// TIA Portal V18 export
FUNCTION_BLOCK "Source_select"   // FB1, FBD
TITLE = Source selection
{ S7_Optimized_Access := 'TRUE' }
VERSION : 0.1
// Source select
// stored: AutoNumber true, IsIECCheckEnabled false, IsRetainMemResEnabled false, MemoryReserve 100, SetENOAutomatically false, UDAEnableTagReadback false
   VAR_INPUT
      START : Bool;
      SP : Real;
      PV : Real;
      COUNTER_SP : Real;
      CHW_CT_SP : Real;
      CT_HW_SP : Real;
      HW_STEAM_SP : Real;
      CT_CHW_SP : Real;
      CHW_CHBr_SP : Real;
   END_VAR
   VAR_OUTPUT
      SOURCE_SEL : Int;
      STATUS : Word;
   END_VAR
   VAR
      Heating : Int;
      Cooling : Int;
      SUB_SP_COUNTER_SP : Real;
      ADD_SP_COUNTER_SP : Real;
      SS_TP1 { S7_SetPoint := 'True'} : TP_TIME;
      SS_TP2 { S7_SetPoint := 'True'} : TP_TIME;
      SS_TP3 { S7_SetPoint := 'True'} : TP_TIME;
      SS_TP4 { S7_SetPoint := 'True'} : TP_TIME;
      SS_TP5 { S7_SetPoint := 'True'} : TP_TIME;
      SS_TP6 { S7_SetPoint := 'True'} : TP_TIME;
      SS_TON1 { S7_SetPoint := 'True'} : TON_TIME;
      SS_TON3 { S7_SetPoint := 'True'} : TON_TIME;
      SS_TON4 { S7_SetPoint := 'True'} : TON_TIME;
      SS_TON5 { S7_SetPoint := 'True'} : TON_TIME;
      SS_TON6 { S7_SetPoint := 'True'} : TON_TIME;
      SS_TON7 { S7_SetPoint := 'True'} : TON_TIME;
   END_VAR
BEGIN

REGION Network 1: Heating
   // Heating
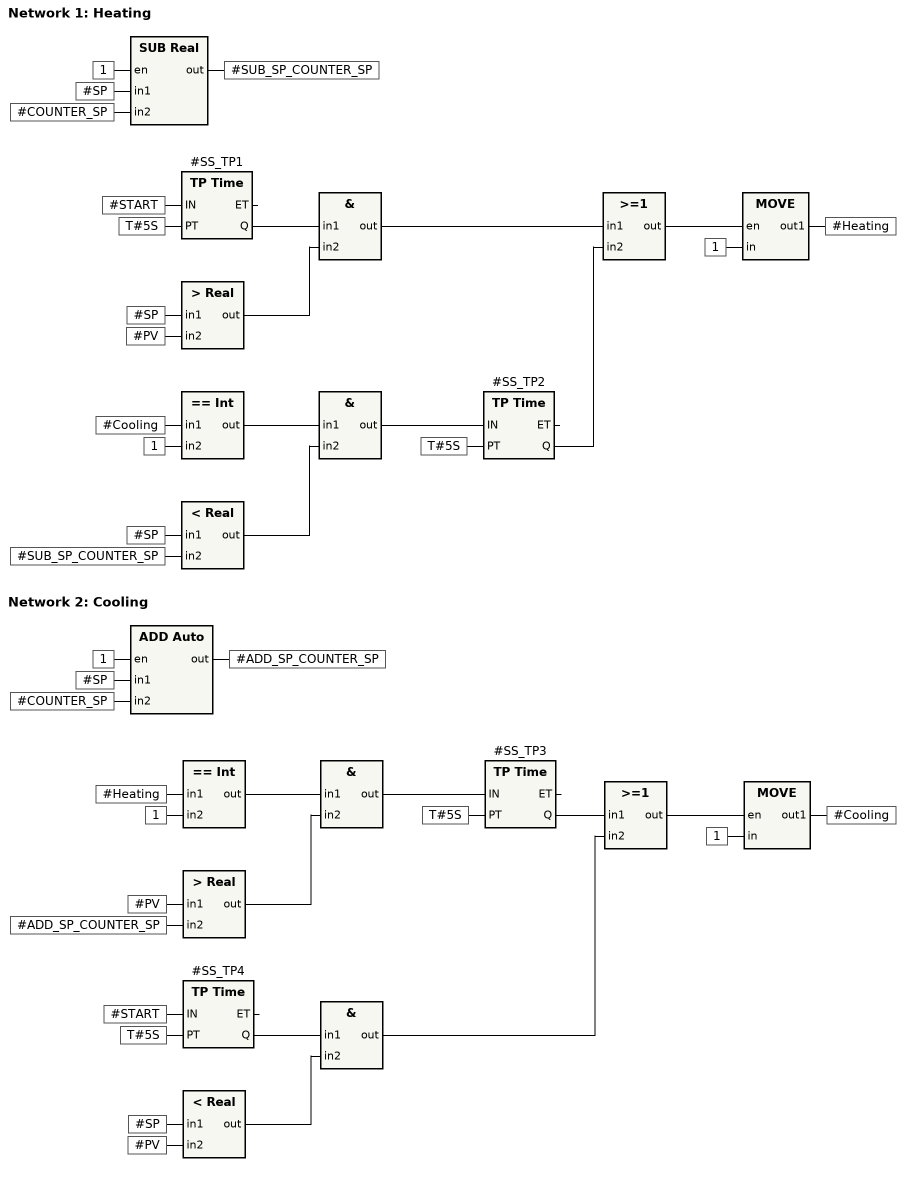
   IF 1 THEN #SUB_SP_COUNTER_SP := #SP - #COUNTER_SP; END_IF;
   #SS_TP1(IN := #START, PT := T#5S);   // TP
   #SS_TP2(IN := (#Cooling = 1) AND (#SP < #SUB_SP_COUNTER_SP), PT := T#5S);   // TP
   IF (#SS_TP1.Q AND (#SP > #PV)) OR #SS_TP2.Q THEN #Heating := 1; END_IF;
END_REGION

REGION Network 2: Cooling
   // Cooling
   IF 1 THEN #ADD_SP_COUNTER_SP := #SP + #COUNTER_SP; END_IF;
   #SS_TP3(IN := (#Heating = 1) AND (#PV > #ADD_SP_COUNTER_SP), PT := T#5S);   // TP
   #SS_TP4(IN := #START, PT := T#5S);   // TP
   IF #SS_TP3.Q OR (#SS_TP4.Q AND (#SP < #PV)) THEN #Cooling := 1; END_IF;
END_REGION

REGION Network 3: Heating & Cooling Reset
   // Heating & Cooling Reset
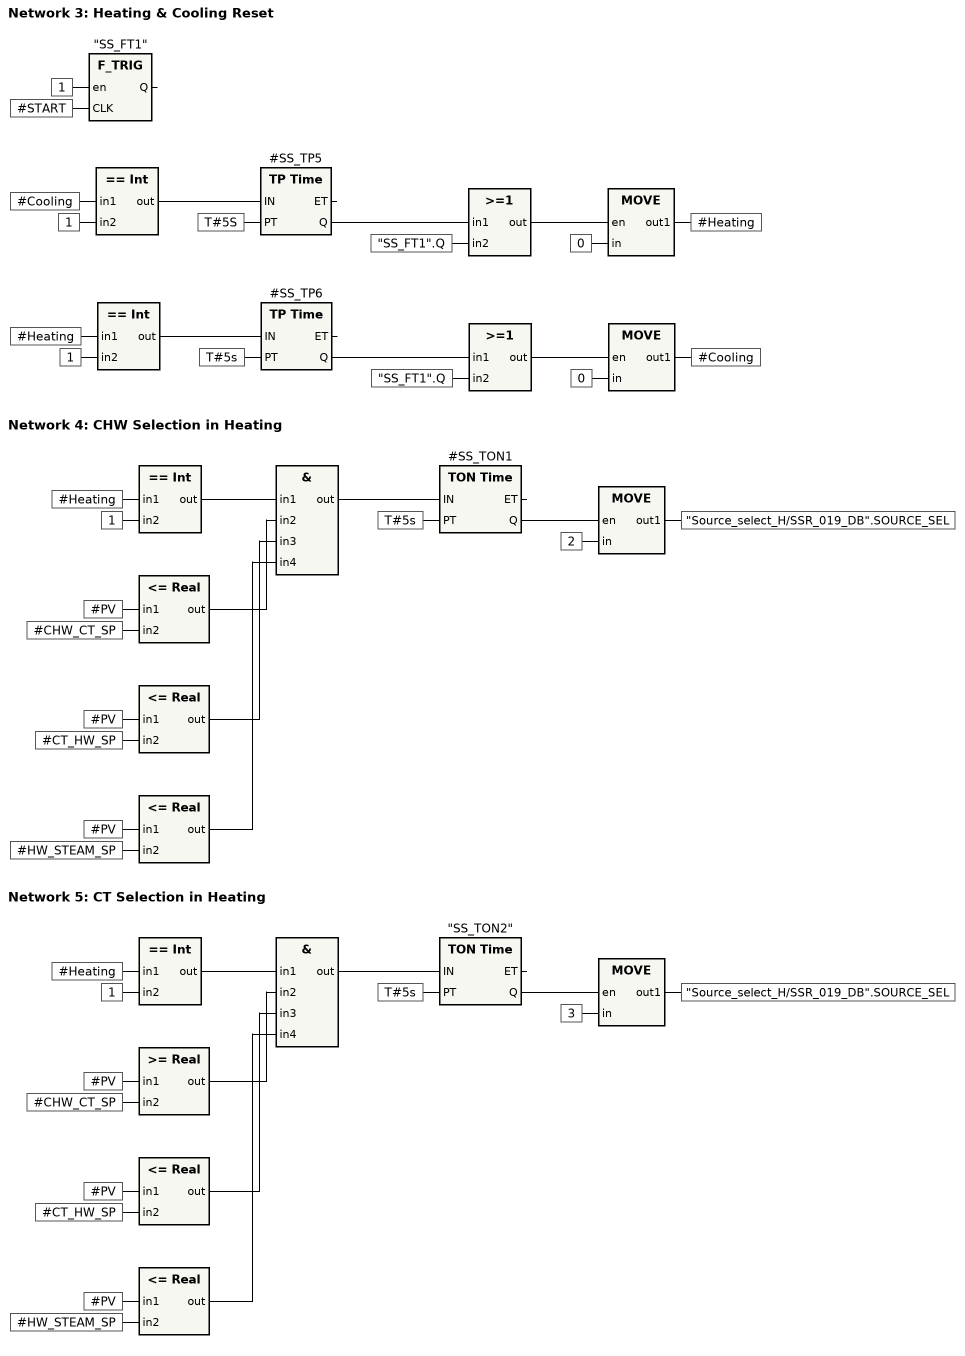
   IF 1 THEN
       "SS_FT1"(CLK := #START);   // F_TRIG
   END_IF;
   #SS_TP5(IN := #Cooling = 1, PT := T#5S);   // TP
   IF #SS_TP5.Q OR "SS_FT1".Q THEN #Heating := 0; END_IF;
   #SS_TP6(IN := #Heating = 1, PT := T#5s);   // TP
   IF #SS_TP6.Q OR "SS_FT1".Q THEN #Cooling := 0; END_IF;
END_REGION

REGION Network 4: CHW Selection in Heating
   // CHW Selection in Heating
   #SS_TON1(IN := (#Heating = 1) AND (#PV <= #CHW_CT_SP) AND (#PV <= #CT_HW_SP) AND (#PV <= #HW_STEAM_SP),   // TON
            PT := T#5s);
   IF #SS_TON1.Q THEN "Source_select_H/SSR_019_DB".SOURCE_SEL := 2; END_IF;
END_REGION

REGION Network 5: CT Selection in Heating
   // CT Selection in Heating
   "SS_TON2".TON(IN := (#Heating = 1) AND (#PV >= #CHW_CT_SP) AND (#PV <= #CT_HW_SP) AND (#PV <= #HW_STEAM_SP),
                 PT := T#5s);
   IF "SS_TON2".Q THEN "Source_select_H/SSR_019_DB".SOURCE_SEL := 3; END_IF;
END_REGION

REGION Network 6: HW Selection in Heating
   // HW Selection in Heating
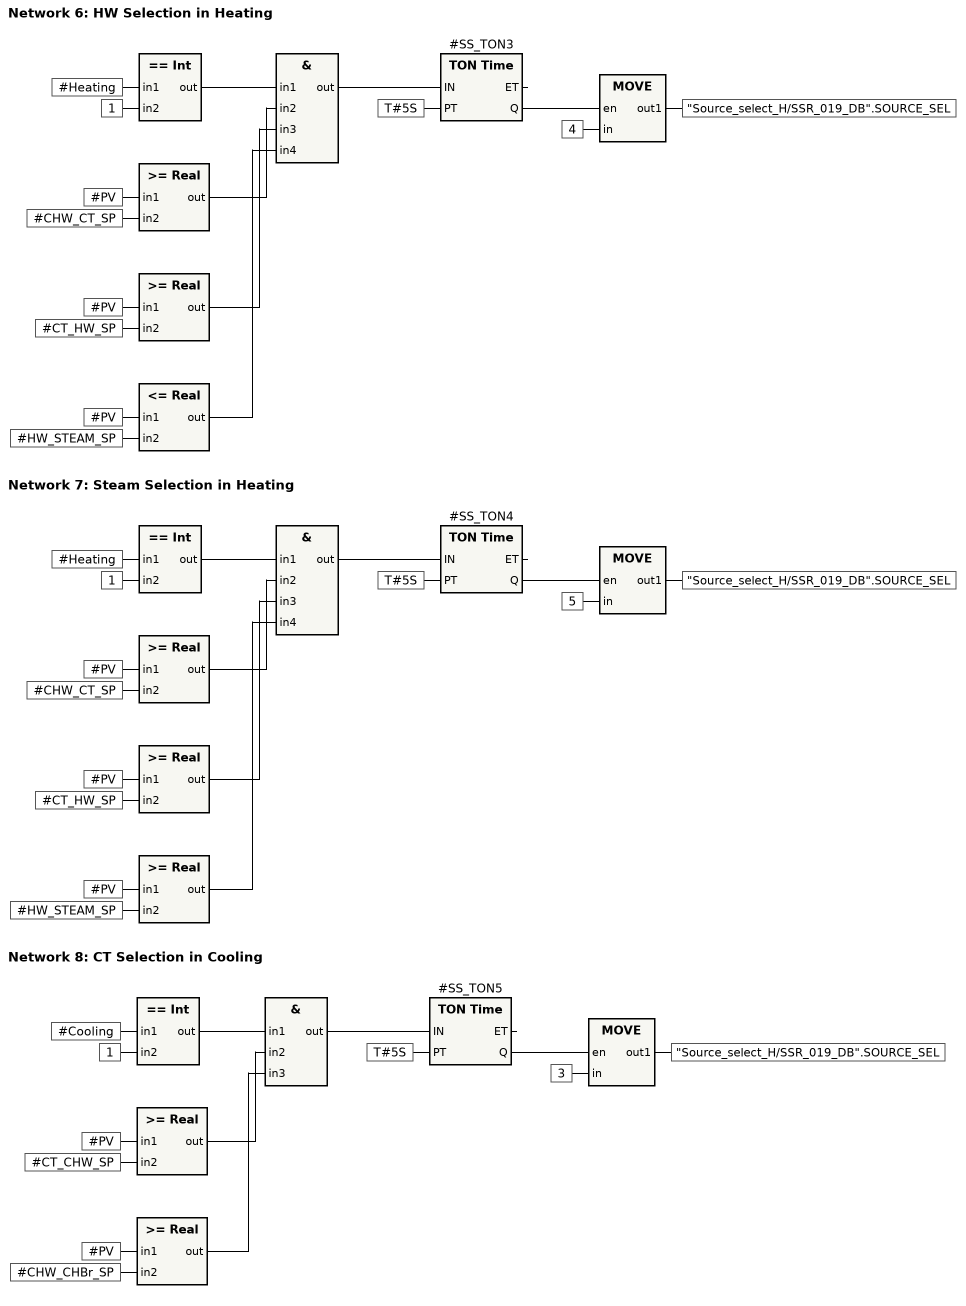
   #SS_TON3(IN := (#Heating = 1) AND (#PV >= #CHW_CT_SP) AND (#PV >= #CT_HW_SP) AND (#PV <= #HW_STEAM_SP),   // TON
            PT := T#5S);
   IF #SS_TON3.Q THEN "Source_select_H/SSR_019_DB".SOURCE_SEL := 4; END_IF;
END_REGION

REGION Network 7: Steam Selection in Heating
   // Steam Selection in Heating
   #SS_TON4(IN := (#Heating = 1) AND (#PV >= #CHW_CT_SP) AND (#PV >= #CT_HW_SP) AND (#PV >= #HW_STEAM_SP),   // TON
            PT := T#5S);
   IF #SS_TON4.Q THEN "Source_select_H/SSR_019_DB".SOURCE_SEL := 5; END_IF;
END_REGION

REGION Network 8: CT Selection in Cooling
   // CT Selection in Cooling
   #SS_TON5(IN := (#Cooling = 1) AND (#PV >= #CT_CHW_SP) AND (#PV >= #CHW_CHBr_SP), PT := T#5S);   // TON
   IF #SS_TON5.Q THEN "Source_select_H/SSR_019_DB".SOURCE_SEL := 3; END_IF;
END_REGION

REGION Network 9: CHW Selection in Cooling
   // CHW Selection in Cooling
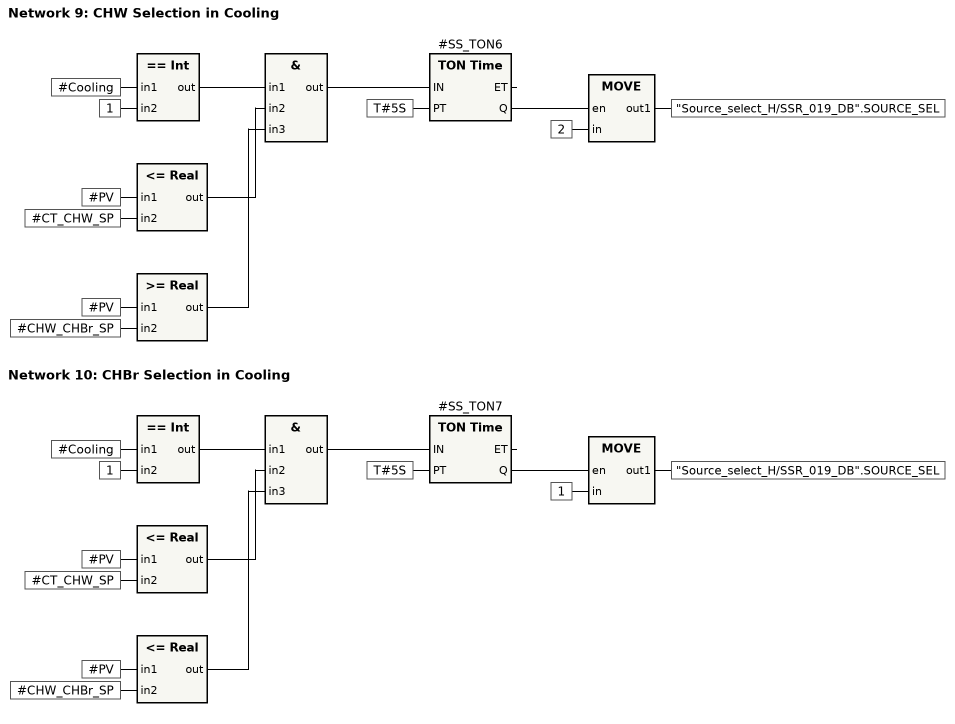
   #SS_TON6(IN := (#Cooling = 1) AND (#PV <= #CT_CHW_SP) AND (#PV >= #CHW_CHBr_SP), PT := T#5S);   // TON
   IF #SS_TON6.Q THEN "Source_select_H/SSR_019_DB".SOURCE_SEL := 2; END_IF;
END_REGION

REGION Network 10: CHBr Selection in Cooling
   // CHBr Selection in Cooling
   #SS_TON7(IN := (#Cooling = 1) AND (#PV <= #CT_CHW_SP) AND (#PV <= #CHW_CHBr_SP), PT := T#5S);   // TON
   IF #SS_TON7.Q THEN "Source_select_H/SSR_019_DB".SOURCE_SEL := 1; END_IF;
END_REGION
END_FUNCTION_BLOCK
